// TwinCAT 3 PLC project PLC01
// ProgramVersion: 3.1.4024.0
// libraries:
//   Tc2_Standard, * (Beckhoff Automation GmbH)
//   Tc2_System, * (Beckhoff Automation GmbH)
//   Tc2_Utilities, * (Beckhoff Automation GmbH)
//   Tc3_Database, * (Beckhoff Automation GmbH)
//   Tc3_EventLogger, * (Beckhoff Automation GmbH)
//   Tc3_Module, * (Beckhoff Automation GmbH)
// project tree:
//   DUTs/Database/ ST_DatabasePower.TcDUT
//   DUTs/HMI/ ST_Valve.TcDUT
//   DUTs/PowerMeter/ ST_AuxConvertedMeasure.TcDUT, ST_AuxiliaryPowerValues.TcDUT, ST_Channel.TcDUT, ST_ConvertedPower.TcDUT, ST_PowerMeter.TcDUT
//   DUTs/ ST_Convert.TcDUT
//   FBs/Database/General/ FB_SQL_ExecuteComandWithoutReturn.TcPOU, FB_SQL_ReadWithData.TcPOU, FB_SQL_TO_CSV.TcPOU
//   FBs/Database/PowerMeter/ FB_SQL_ReadPower.TcPOU, FB_SQL_WritePower.TcPOU
//   FBs/PowerMeter/ FB_LastTimeSimple.TcPOU, FB_MeasureAuxPhasePower.TcPOU, FB_PowerMeter.TcPOU, FB_Simulate_EL3433.TcPOU
//   FBs/Process/ FB_Pump.TcPOU, FB_Valve.TcPOU
//   FCs/ FC_ConcatStr.TcPOU
//   GVLs/ GVL.TcGVL, GVL_HMI.TcGVL, GVL_IO.TcGVL
//   / PlcTask.TcTTO
//   POUs/Database/ PRG_Database.TcPOU
//   POUs/Eletric/ PRG_Eletric.TcPOU
//   POUs/ MAIN.TcPOU
//   POUs/PowerMeter/ PRG_PowerMeter.TcPOU
//   POUs/Process/ PRG_Process.TcPOU
// real-time tasks:
//   TASK PlcTask: cycle T#10ms, priority 20, ADS port 350
// motion (NC):
//   TASK NC-Task 1 SAF: cycle T#2ms, priority 4, ADS port 501
//   TASK NC-Task 1 SVB: cycle T#10ms, priority 8, ADS port 511
//   AXIS Eixo X (id 1)
//     OtherSettings: AllowMotionCmdToSlave=true
//     encoder EncType=1
//     drive DrvType=5
//       Analog: TorqueSetpointScale=10, ScaleFactorActTorque=0.1
//     controller CtrType=1
//       CtrPara: PriorControlFactor=1
//         Observer: BandWidth=20
// I/O:
//   DEVICE Device 3 (EtherCAT), AmsNetId 169.254.242.29.4.1
//     Term 1 (EK1100) [EK1100 EtherCAT Coupler (2A E-Bus)]
//       Term 2 (EL1008) [EL1008 8Ch. Dig. Input 24V, 3ms]
//       Term 3 (EL2008) [EL2008 8Ch. Dig. Output 24V, 0.5A]
//       Term 4 (EL3062) [EL3062 2Ch. Ana. Input 0-10V]
//       Term 5 (EL4002) [EL4002 2Ch. Ana. Output 0-10V, 12bit]
//       Term 6 (EL3433) [EL3433 3Ch. Power Measuring]
//       Term 7 (EL6900) [EL6900, TwinSAFE PLC]
//       Term 8 (EK1310) [EK1310 EtherCAT P extension with feed-in]
// variable links:
//   PLC01/PLC01 Instance <-> Device 3 (EtherCAT)/Term 1 (EK1100)/Term 6 (EL3433)
//     PlcTask Inputs/PRG_PowerMeter.EL3433_Ch1/ActivePower <-> PM Inputs Channel 1/Active power
//     PlcTask Inputs/PRG_PowerMeter.EL3433_Ch2/ActivePower <-> PM Inputs Channel 2/Active power
//     PlcTask Inputs/PRG_PowerMeter.EL3433_Ch3/ActivePower <-> PM Inputs Channel 3/Active power
//     PlcTask Inputs/PRG_PowerMeter.EL3433_Ch1/Current <-> PM Inputs Channel 1/Current
//     PlcTask Inputs/PRG_PowerMeter.EL3433_Ch2/Current <-> PM Inputs Channel 2/Current
//     PlcTask Inputs/PRG_PowerMeter.EL3433_Ch3/Current <-> PM Inputs Channel 3/Current
//     PlcTask Inputs/PRG_PowerMeter.EL3433_Ch1/Index <-> PM Inputs Channel 1/Index
//     PlcTask Inputs/PRG_PowerMeter.EL3433_Ch2/Index <-> PM Inputs Channel 2/Index
//     PlcTask Inputs/PRG_PowerMeter.EL3433_Ch3/Index <-> PM Inputs Channel 3/Index
//     PlcTask Inputs/PRG_PowerMeter.EL3433_Ch1/Status/MissingZeroCrossing <-> PM Inputs Channel 1/STATUS/Missing zero crossing
//     PlcTask Inputs/PRG_PowerMeter.EL3433_Ch2/Status/MissingZeroCrossing <-> PM Inputs Channel 2/STATUS/Missing zero crossing
//     PlcTask Inputs/PRG_PowerMeter.EL3433_Ch3/Status/MissingZeroCrossing <-> PM Inputs Channel 3/STATUS/Missing zero crossing
//     PlcTask Inputs/PRG_PowerMeter.EL3433_Ch1/Status/OverCurrent <-> PM Inputs Channel 1/STATUS/Overcurrent
//     PlcTask Inputs/PRG_PowerMeter.EL3433_Ch2/Status/OverCurrent <-> PM Inputs Channel 2/STATUS/Overcurrent
//     PlcTask Inputs/PRG_PowerMeter.EL3433_Ch3/Status/OverCurrent <-> PM Inputs Channel 3/STATUS/Overcurrent
//     PlcTask Inputs/PRG_PowerMeter.EL3433_Ch1/Status/OverVoltage <-> PM Inputs Channel 1/STATUS/Overvoltage
//     PlcTask Inputs/PRG_PowerMeter.EL3433_Ch2/Status/OverVoltage <-> PM Inputs Channel 2/STATUS/Overvoltage
//     PlcTask Inputs/PRG_PowerMeter.EL3433_Ch3/Status/OverVoltage <-> PM Inputs Channel 3/STATUS/Overvoltage
//     PlcTask Inputs/PRG_PowerMeter.EL3433_Ch1/Status/PhaseSeqCCW <-> PM Inputs Channel 1/STATUS/Phase sequence ccw
//     PlcTask Inputs/PRG_PowerMeter.EL3433_Ch2/Status/PhaseSeqCCW <-> PM Inputs Channel 2/STATUS/Phase sequence ccw
//     PlcTask Inputs/PRG_PowerMeter.EL3433_Ch3/Status/PhaseSeqCCW <-> PM Inputs Channel 3/STATUS/Phase sequence ccw
//     PlcTask Inputs/PRG_PowerMeter.EL3433_Ch1/Status/PhaseSeqCW <-> PM Inputs Channel 1/STATUS/Phase sequence cw
//     PlcTask Inputs/PRG_PowerMeter.EL3433_Ch2/Status/PhaseSeqCW <-> PM Inputs Channel 2/STATUS/Phase sequence cw
//     PlcTask Inputs/PRG_PowerMeter.EL3433_Ch3/Status/PhaseSeqCW <-> PM Inputs Channel 3/STATUS/Phase sequence cw
//     PlcTask Inputs/PRG_PowerMeter.EL3433_Ch1/Status/TxPdoState <-> PM Inputs Channel 1/STATUS/TxPDO State
//     PlcTask Inputs/PRG_PowerMeter.EL3433_Ch2/Status/TxPdoState <-> PM Inputs Channel 2/STATUS/TxPDO State
//     PlcTask Inputs/PRG_PowerMeter.EL3433_Ch3/Status/TxPdoState <-> PM Inputs Channel 3/STATUS/TxPDO State
//     PlcTask Inputs/PRG_PowerMeter.EL3433_Ch1/Status/TxPdoToggle <-> PM Inputs Channel 1/STATUS/TxPDO Toggle
//     PlcTask Inputs/PRG_PowerMeter.EL3433_Ch2/Status/TxPdoToggle <-> PM Inputs Channel 2/STATUS/TxPDO Toggle
//     PlcTask Inputs/PRG_PowerMeter.EL3433_Ch3/Status/TxPdoToggle <-> PM Inputs Channel 3/STATUS/TxPDO Toggle
//     PlcTask Inputs/PRG_PowerMeter.EL3433_Ch1/Status/UnderVoltage <-> PM Inputs Channel 1/STATUS/Undervoltage
//     PlcTask Inputs/PRG_PowerMeter.EL3433_Ch2/Status/UnderVoltage <-> PM Inputs Channel 2/STATUS/Undervoltage
//     PlcTask Inputs/PRG_PowerMeter.EL3433_Ch3/Status/UnderVoltage <-> PM Inputs Channel 3/STATUS/Undervoltage
//     PlcTask Inputs/PRG_PowerMeter.EL3433_Ch1/VariantValue <-> PM Inputs Channel 1/Variant value
//     PlcTask Inputs/PRG_PowerMeter.EL3433_Ch2/VariantValue <-> PM Inputs Channel 2/Variant value
//     PlcTask Inputs/PRG_PowerMeter.EL3433_Ch3/VariantValue <-> PM Inputs Channel 3/Variant value
//     PlcTask Inputs/PRG_PowerMeter.EL3433_Ch1/Voltage <-> PM Inputs Channel 1/Voltage
//     PlcTask Inputs/PRG_PowerMeter.EL3433_Ch2/Voltage <-> PM Inputs Channel 2/Voltage
//     PlcTask Inputs/PRG_PowerMeter.EL3433_Ch3/Voltage <-> PM Inputs Channel 3/Voltage
//     PlcTask Outputs/PRG_PowerMeter.Ch1_OutIndex <-> PM Outputs Channel 1/Index
//     PlcTask Outputs/PRG_PowerMeter.Ch2_OutIndex <-> PM Outputs Channel 2/Index
//     PlcTask Outputs/PRG_PowerMeter.Ch3_OutIndex <-> PM Outputs Channel 3/Index
//     PlcTask Outputs/PRG_PowerMeter.ChAux_OutIndex <-> PM Outputs Auxiliary/Index

CONFIGURATION PLC01
    RESOURCE PLC ON TwinCAT3
        TASK PlcTask(INTERVAL := T#10ms, PRIORITY := 20);
        PROGRAM MAIN WITH PlcTask : MAIN;
    END_RESOURCE
END_CONFIGURATION

// ---- DUTs/Database/ST_DatabasePower.TcDUT
TYPE ST_DatabasePower :
STRUCT
	ID 					: T_ULARGE_INTEGER  ;	//IDENTITY
	Timestamp 			: DATE_AND_TIME ;		//TIMESTAMP
	Name 				: STRING(50) ;			//NAME OF LOAD
	ActivePower 		: LREAL ;				//ACTIVE POWER
	ApparentPower 		: LREAL ;				//APARENT POWER
	ReactivePower 		: LREAL ;				//REACTIVE POWER
	Voltage 			: LREAL ;				//VOLTAGE
	Current 			: LREAL ;				//CURRENT
	Cosphi				: LREAL	;				//COSENO PHI
	Frequency			: LREAL	;				//FREQUENCY
	AngleBetweenPhase1	: LREAL	;				//ANGLE BETWEEN FASE 1	
	Energy 				: LREAL ;				//POSITIVE ENERGY
	EnergyNegative		: LREAL	;				//NEGATIVE ENERGY
END_STRUCT
END_TYPE

// ---- DUTs/HMI/ST_Valve.TcDUT
TYPE ST_Valve :
STRUCT
	status : BOOL ;
	comando : BOOL ;
	auto_manual : BOOL ;
	time_feedback : INT ;
END_STRUCT
END_TYPE

// ---- DUTs/PowerMeter/ST_AuxConvertedMeasure.TcDUT
TYPE ST_AuxConvertedMeasure :
	STRUCT
		sumOfEnergy : LREAL;									//index 2. 
		frequency : LREAL;										//4
		sumOfEnergyNeg : LREAL;									//5
		sumOfActivePower : LREAL;								//10
		sumOfApparentPower : LREAL;								//11
		sumOfReactivePower : LREAL;								//12
		adcTemp : LREAL ;										//100
		aHarmonicCurrentValue : ARRAY[1..3,1..21] OF LREAL;		//
		aHarmonicCurrentRatio : ARRAY[1..3,1..21] OF LREAL;		//
		aHarmonicVoltageValue : ARRAY[1..3,1..21] OF LREAL;		//
		aHarmonicVoltageRatio : ARRAY[1..3,1..21] OF LREAL;		//
		aAuxPowerValues : ARRAY[1..3] OF ST_ConvertedPower;		//
	END_STRUCT
END_TYPE

// ---- DUTs/PowerMeter/ST_AuxiliaryPowerValues.TcDUT
TYPE ST_AuxiliaryPowerValues :
	STRUCT
		index:USINT;		//Indice
		channel:USINT;		//Canal
		value:DINT;			//Valor
	END_STRUCT
END_TYPE

// ---- DUTs/PowerMeter/ST_Channel.TcDUT
TYPE ST_Channel :
	STRUCT
		OverVoltage : BIT ; //
		UnderVoltage : BIT ; //
		OverCurrent : BIT ; //
		PhaseSeqCW : BIT ; //
		PhaseSeqCCW : BIT ; //
		MissingZeroCrossing : BIT ; //
		TxPdoState : BIT ; //
		TxPdoToggle : BIT ; //
	END_STRUCT
END_TYPE

// ---- DUTs/PowerMeter/ST_ConvertedPower.TcDUT
TYPE ST_ConvertedPower :
	STRUCT
		Current			:LREAL	;	//Display the channel's current 
		Voltage			:LREAL	;	//Display the channel's voltage
		ActivePower		:LREAL	;	//Display the channel's active power
		ApparentPower	:LREAL	;	//Potência aparente
		ReactivePower	:LREAL	;	//potencia reativa
		Energy			:LREAL	;	//Energia
		Cosphi			:LREAL	;	//cosseno PHI
		Frequency		:LREAL	;	//Display the channel's Frequency
		EnergyNegative	:LREAL	;	//Energia (Negativa)
		AngleBetweenPhase1	:LREAL	;	//Angulo entre essa fase e a fase 1
	END_STRUCT
END_TYPE

// ---- DUTs/PowerMeter/ST_PowerMeter.TcDUT
TYPE ST_PowerMeter :
	STRUCT
		Status 			: ST_Channel ; 	//Todos os status de cada canal (Overvoltage, UnderVoltage, Overcurrent, PhaseSequenceZero Crossing...)
		Current 		: DINT ; 		//
		Voltage 		: DINT ; 		//
		ActivePower 	: DINT ; 		//
		Index 			: USINT ; 		//
		VariantValue	: DINT ; 		//
	END_STRUCT
END_TYPE

// ---- DUTs/ST_Convert.TcDUT
TYPE ST_Convert :
UNION
	aWORD : ARRAY[0..10] OF INT ;
	aREAL : ARRAY[0..5] OF REAL ;
END_UNION
END_TYPE

// ---- GVLs/GVL.TcGVL
{attribute 'qualified_only'}
VAR_GLOBAL
	(* Estruturas com os valores convertidos *)	
	EL3433_Ch1_PowerConverted : ST_ConvertedPower; //Estrutura que retorna os valores da Fase 1 (Tensao, Corrente...)
	EL3433_Ch2_PowerConverted : ST_ConvertedPower; //Estrutura que retorna os valores da Fase 1 (Tensao, Corrente...)
	EL3433_Ch3_PowerConverted : ST_ConvertedPower; //Estrutura que retorna os valores da Fase 1 (Tensao, Corrente...)
END_VAR

// ---- GVLs/GVL_HMI.TcGVL
{attribute 'qualified_only'}
VAR_GLOBAL
	DateStart : STRING ;
	DateEnd : STRING ;
END_VAR

// ---- GVLs/GVL_IO.TcGVL
{attribute 'qualified_only'}
VAR_GLOBAL


END_VAR

// ---- POUs/MAIN.TcPOU
PROGRAM MAIN
VAR
	stMyTest : ST_Convert ;

END_VAR



PRG_PowerMeter() ;

PRG_Database();

END_PROGRAM

// ---- POUs/PowerMeter/PRG_PowerMeter.TcPOU
PROGRAM PRG_PowerMeter
VAR	

(* Seleciona vaores REAIS do EL3433 ou Simulados *)
	bSelectValues : BOOL ;

(* Bloco para simulacao de valores do EL3433 *)
	fbPowerL1Simulate : FB_Simulate_EL3433 ;
	fbPowerL2Simulate : FB_Simulate_EL3433 ;
	fbPowerL3Simulate : FB_Simulate_EL3433 ;

(* Blocos de funcao para cada canal do terminal EL3433 REAL *)	
	fbPowerL1 : FB_PowerMeter ; //Bloco para extratir os dados do cartão
	fbPowerL2 : FB_PowerMeter ; //Bloco para extratir os dados do cartão
	fbPowerL3 : FB_PowerMeter ; //Bloco para extratir os dados do cartão
	fbAuxPower : FB_MeasureAuxPhasePower ; //	
	
(* Estruturas com link com o IO EL3433*)
	EL3433_Ch1 AT %I* : ST_PowerMeter ;
	EL3433_Ch2 AT %I* : ST_PowerMeter ;
	EL3433_Ch3 AT %I* : ST_PowerMeter ;	

(* Variavel Index do terminal EL3433 *)
	Ch1_OutIndex AT %Q*: USINT := 0 ;
	Ch2_OutIndex AT %Q*: USINT := 0 ;
	Ch3_OutIndex AT %Q*: USINT := 0 ;
	ChAux_OutIndex AT %Q*: USINT := 0 ;	
	

	stConvertedAuxChn : ST_AuxConvertedMeasure; //	
	
END_VAR


IF bSelectValues = FALSE THEN
	
	fbPowerL1Simulate(
		bExecute:= TRUE, 
		Current=> GVL.EL3433_Ch1_PowerConverted.Current, 
		Voltage=> GVL.EL3433_Ch1_PowerConverted.Voltage, 
		ActivePower=> GVL.EL3433_Ch1_PowerConverted.ActivePower, 
		ApparentPower=> GVL.EL3433_Ch1_PowerConverted.ApparentPower, 
		ReactivePower=> GVL.EL3433_Ch1_PowerConverted.ReactivePower, 
		Energy=> GVL.EL3433_Ch1_PowerConverted.Energy, 
		Cosphi=> GVL.EL3433_Ch1_PowerConverted.Cosphi, 
		Frequency=> GVL.EL3433_Ch1_PowerConverted.Frequency, 
		EnergyNegative=> GVL.EL3433_Ch1_PowerConverted.EnergyNegative, 
		AngleBetweenPhase1=> GVL.EL3433_Ch1_PowerConverted.AngleBetweenPhase1);
		
		
		GVL.EL3433_Ch2_PowerConverted := GVL.EL3433_Ch1_PowerConverted;
		GVL.EL3433_Ch3_PowerConverted := GVL.EL3433_Ch1_PowerConverted;
ELSE

	fbPowerL1(PowerInput:= EL3433_Ch1, PowerConverted=> GVL.EL3433_Ch1_PowerConverted, OutIndex=> Ch1_OutIndex);
	fbPowerL2(PowerInput:= EL3433_Ch2, PowerConverted=> GVL.EL3433_Ch2_PowerConverted, OutIndex=> Ch2_OutIndex);
	fbPowerL3(PowerInput:= EL3433_Ch3, PowerConverted=> GVL.EL3433_Ch3_PowerConverted, OutIndex=> Ch3_OutIndex);
	fbAuxPower(convertedMeasure=> stConvertedAuxChn);


END_IF

END_PROGRAM

// ---- FBs/PowerMeter/FB_Simulate_EL3433.TcPOU
FUNCTION_BLOCK FB_Simulate_EL3433
VAR_INPUT
	bExecute : BOOL ;
END_VAR
VAR_OUTPUT
	Current			:LREAL	;	//Display the channel's current 
	Voltage			:LREAL	;	//Display the channel's voltage
	ActivePower		:LREAL	;	//Display the channel's active power
	ApparentPower	:LREAL	;	//Potência aparente
	ReactivePower	:LREAL	;	//potencia reativa
	Energy			:LREAL	;	//Energia
	Cosphi			:LREAL	;	//cosseno PHI
	Frequency		:LREAL	;	//Display the channel's Frequency
	EnergyNegative	:LREAL	;	//Energia (Negativa)
	AngleBetweenPhase1	:LREAL	;	//Angulo entre essa fase e a fase 1
END_VAR
VAR
    tCurrentTime: TIME;
    rRandomValue: REAL;
	fRandom : DRAND ;
END_VAR


   fRandom(Seed:= 1 , Num=> rRandomValue);  // Converte o tempo atual para milissegundos

IF bExecute = TRUE THEN 

	Current			:=	rRandomValue + 2;	//Display the channel's current 
	Voltage			:=	rRandomValue + 379;	//Display the channel's voltage
	Cosphi			:=	(rRandomValue + 81) * 0.01;		
	ActivePower		:=	Voltage * Current * Cosphi;	//Display the channel's active power
	ApparentPower	:=	Voltage * Current;	//Potência aparente
	ReactivePower	:=	Voltage * Current * SQRT( 1 - Cosphi * Cosphi) ;	//potencia reativa
	Energy			:=	rRandomValue * 10;	
	Frequency		:=	rRandomValue + 59;	
	EnergyNegative	:=	rRandomValue * 10;	
	AngleBetweenPhase1	:=	rRandomValue + 60;	
END_IF

END_FUNCTION_BLOCK

// ---- FBs/PowerMeter/FB_PowerMeter.TcPOU
FUNCTION_BLOCK FB_PowerMeter
VAR_INPUT
	PowerInput : ST_PowerMeter;	
END_VAR
VAR_OUTPUT
	PowerConverted : ST_ConvertedPower;	//Valores convertidos
	OutIndex : USINT :=0;	
END_VAR
VAR
	iAux:UINT:=0;
END_VAR

(* Conversao da corrente *)
powerConverted.current:=DINT_TO_LREAL(PowerInput.current)*0.000001;

(* Conversao da Tensao *)
powerConverted.voltage:=DINT_TO_LREAL(PowerInput.voltage)*0.0001;

(* Conversao da potencia ativa *)
powerConverted.activePower:=DINT_TO_LREAL(PowerInput.activePower)*0.01;

(* Conversoes diversas *)

CASE PowerInput.index OF
	0:
		powerConverted.apparentPower := DINT_TO_LREAL(PowerInput.variantValue) * 0.01 ;
	1:
		powerConverted.reactivePower := DINT_TO_LREAL(PowerInput.variantValue) * 0.01 ;
	2:
		powerConverted.energy := DINT_TO_LREAL(PowerInput.variantValue) * 0.001;
	3:
		powerConverted.cosphi := DINT_TO_LREAL(PowerInput.variantValue) * 0.001;
	4:
		powerConverted.frequency := DINT_TO_LREAL(PowerInput.variantValue) * 0.1;
	5:
		powerConverted.energy := DINT_TO_LREAL(PowerInput.variantValue) * 0.001 ;
	6:
		powerConverted.AngleBetweenPhase1 := DINT_TO_LREAL(PowerInput.variantValue) * 0.01;
END_CASE

IF (PowerInput.index = OutIndex)THEN
	iAux := iAux + 1 ;
	IF iAux > 4 THEN
		iAux := 0 ;
		IF outIndex <= 6 THEN
			outIndex := outIndex + 1 ;
		ELSE
			outIndex := 0 ;	
		END_IF
	END_IF	
END_IF

END_FUNCTION_BLOCK

// ---- FBs/PowerMeter/FB_MeasureAuxPhasePower.TcPOU
FUNCTION_BLOCK FB_MeasureAuxPhasePower
VAR_INPUT
END_VAR
VAR_OUTPUT
	convertedMeasure:ST_AuxConvertedMeasure;
	tLastHarmonicMeasureTime:TIME;
	lastiTime:FB_LastTimeSimple;
END_VAR
VAR
	power AT %I*:ST_AuxiliaryPowerValues;
	iChannel AT %Q*:USINT;
	iIndex AT %Q*:USINT;
	bMeasureTime:BOOL;
END_VAR

CASE power.channel OF
	0:
		CASE power.index OF
			0:
				iIndex := 2 ;
			2:
				convertedMeasure.sumOfEnergy := DINT_TO_LREAL(power.value) * 0.001;
				iIndex:=4;
				//F_DebugCount(1);
			4:
				convertedMeasure.frequency := DINT_TO_LREAL(power.value) * 0.1;
				iIndex:=5;
				//F_DebugCount(2);
			5:
				convertedMeasure.sumOfEnergyNeg := DINT_TO_LREAL(power.value) * 0.001;
				iIndex:=10;
				//F_DebugCount(3);				
			10:
				convertedMeasure.sumOfActivePower := DINT_TO_LREAL(power.value) * 0.01;
				iIndex:=11;
				//F_DebugCount(4);
			11:
				convertedMeasure.sumOfApparentPower := DINT_TO_LREAL(power.value)*0.01;
				iIndex:=12;
				//F_DebugCount(5);				
			12:
				convertedMeasure.sumOfReactivePower := DINT_TO_LREAL(power.value)*0.01;
				iIndex:=100;
				//F_DebugCount(6);				
			100:
				convertedMeasure.adcTemp := DINT_TO_LREAL(power.value);
				iIndex:=1;
				iChannel:=1;
				bMeasureTime:=TRUE;	//Inicia o tempo de leitura das harmonicas
				//F_DebugCount(7);
		END_CASE
	1..3:
		CASE power.index OF
			0:
				;
			100:
				;
			1..21:
				convertedMeasure.aHarmonicCurrentValue[power.channel,power.index]:=DINT_TO_LREAL(power.value)*0.000001;
				IF (power.index <21) AND (iIndex < 21) THEN
					iIndex:=iIndex+1;
				ELSIF (power.index = 21 ) AND (power.channel < 3) THEN
					iIndex:=1;
					IF power.channel = iChannel THEN
						iChannel:=iChannel+1;
					END_IF
				ELSIF (power.index = 21) AND (power.channel >=3) THEN
					iChannel:=1;		//Modificar
					iIndex:=51;
				END_IF
			51..71:
				convertedMeasure.aHarmonicCurrentRatio[power.channel,power.index-50]:=DINT_TO_LREAL(power.value)*0.01;
				IF (power.index <71) AND (iIndex < 71) THEN
					iIndex:=iIndex+1;
				ELSIF (power.index = 71 ) AND (power.channel < 3) THEN
					iIndex:=51;
					IF power.channel = iChannel THEN
						iChannel:=iChannel+1;
					END_IF
				ELSIF (power.index = 71) AND (power.channel >=3) THEN
					iChannel:=1;		//Modificar
					iIndex:=101;
				END_IF
			101..121:
				convertedMeasure.aHarmonicVoltageValue[power.channel,power.index-100]:=DINT_TO_LREAL(power.value)*0.0001;
				IF (power.index <121) AND (iIndex < 121) THEN
					iIndex:=iIndex+1;
				ELSIF (power.index = 121 ) AND (power.channel < 3) THEN
					iIndex:=101;
					IF power.channel = iChannel THEN
						iChannel:=iChannel+1;
					END_IF
				ELSIF (power.index = 121) AND (power.channel >=3) THEN
					iChannel:=1;		//Modificar
					iIndex:=151;
				END_IF

			151..171:
				convertedMeasure.aHarmonicVoltageRatio[power.channel,power.index-150]:=DINT_TO_LREAL(power.value)*0.01;
				IF (power.index <171) AND (iIndex < 171) THEN
					iIndex:=iIndex+1;
				ELSIF (power.index = 171 ) AND (power.channel < 3) THEN
					iIndex:=151;
					IF power.channel = iChannel THEN
						iChannel:=iChannel+1;
					END_IF
				ELSIF (power.index = 171) AND (power.channel >=3) THEN
					iChannel:=11;		
					iIndex:=0;
					bMeasureTime:=FALSE;					
				END_IF
			ELSE
				iChannel:=0;
				iIndex:=0;
				bMeasureTime:=FALSE;
		END_CASE
	11..13:
		CASE power.index OF
			0:
				IF iIndex = power.index THEN
					iIndex := iIndex+1;
				END_IF
				convertedMeasure.aAuxPowerValues[power.channel-10].apparentPower := DINT_TO_LREAL(power.value)*0.01;
			1:
				IF iIndex = power.index THEN
					iIndex:=iIndex+1;
				END_IF	
				convertedMeasure.aAuxPowerValues[power.channel-10].reactivePower := DINT_TO_LREAL(power.value)*0.01;
			2:
				IF iIndex = power.index THEN
					iIndex:=iIndex+1;
				END_IF
				convertedMeasure.aAuxPowerValues[power.channel-10].energy := DINT_TO_LREAL(power.value)*0.001;
			3:
				IF iIndex = power.index THEN
					iIndex:=iIndex+1;
				END_IF
				convertedMeasure.aAuxPowerValues[power.channel-10].cosPhi := DINT_TO_LREAL(power.value)*0.001;
			4:
				IF iIndex = power.index THEN
					iIndex:=iIndex+1;
				END_IF
				convertedMeasure.aAuxPowerValues[power.channel-10].frequency := DINT_TO_LREAL(power.value)*0.1;
			5:
				IF iIndex = power.index THEN
					iIndex:=iIndex+1;
				END_IF
				convertedMeasure.aAuxPowerValues[power.channel-10].EnergyNegative := DINT_TO_LREAL(power.value)*0.001;
			6:
				IF iIndex = power.index THEN
					iIndex:=10;
				END_IF
				convertedMeasure.aAuxPowerValues[power.channel-10].AngleBetweenPhase1 := DINT_TO_LREAL(power.value)*0.01;
			10:
				IF iIndex = power.index THEN
					iIndex:=11;
				END_IF
				convertedMeasure.aAuxPowerValues[power.channel-10].current := DINT_TO_LREAL(power.value)*0.000001;
			11:
				IF iIndex = power.index THEN
					iIndex:=12;
				END_IF
				convertedMeasure.aAuxPowerValues[power.channel-10].voltage := DINT_TO_LREAL(power.value)*0.0001;
			12:
				convertedMeasure.aAuxPowerValues[power.channel-10].activePower := DINT_TO_LREAL(power.value)*0.01;
				IF power.channel = 13 THEN
					iIndex:=0;
					iChannel:=0;
				ELSE
					IF iChannel = power.channel AND power.channel < 13 THEN
						iChannel:=iChannel+1;
					END_IF
					iIndex:=0;
				END_IF
		END_CASE
END_CASE
lastiTime(bCountTime:= bMeasureTime, tLastTime=> tLastHarmonicMeasureTime);

END_FUNCTION_BLOCK

// ---- FBs/PowerMeter/FB_LastTimeSimple.TcPOU
FUNCTION_BLOCK FB_LastTimeSimple
VAR_INPUT
	bCountTime:BOOL;
END_VAR
VAR_OUTPUT
	tLastTime:TIME;
END_VAR
VAR
	t1:TON;
	timeCountedF_TRIG:F_TRIG;
	tActualtime:TIME;
END_VAR

IF timeCountedF_TRIG.Q THEN
	tLastTime:=tActualtime;
	tActualtime:=T#0S;
END_IF
timeCountedF_TRIG(CLK:=bCountTime);
t1(IN:= bCountTime, PT:=T#1D);
tActualtime:= MAX(tActualtime,t1.ET);

END_FUNCTION_BLOCK

// ---- POUs/Database/PRG_Database.TcPOU
PROGRAM PRG_Database
VAR
(* CREATE TABLE *)	
	fbCreateTable : FB_SQL_ExecuteComandWithoutReturn ;
	bCreateDatabase : BOOL ;
	bDatabaseCreated : BOOL ;
	sSqlCmdCreateTable : STRING(512) ;
	sError : STRING ;
	
(* CREATE CSV *)	
	fbSqlToCsv : FB_SQL_ExecuteComandWithoutReturn ;	
	sSqlCmdSqlToCsv : STRING(512) ;
	
(* WRITE TO DATABASE *)	
	fbSQLWrite_01 : FB_SQL_WritePower ;
	fbSQLWrite_02 : FB_SQL_WritePower ;
	fbSQLWrite_03 : FB_SQL_WritePower ;	
	bEnableWrite: BOOL := TRUE ;
	
(* READ FROM DATABASE *)	
	fbSQLRead_01 : FB_SQL_ReadPower ;
	

	bExecuteRead: BOOL;


END_VAR

(**********************************************************************************)	
(***************** CRIAR TABELA / CREATE TABLE / CREAR TABLA **********************)

sSqlCmdCreateTable := 'CREATE TABLE [TB_PowerMeter22] ([ID] bigint IDENTITY(1,1), [Timestamp] datetime, [Name] varchar(50), [ActivePower] float, [ApparentPower] float, [ReactivePower] float, [Voltage] float, [Current] float, [Cosphi] float, [Frequency] float, [AngleBetweenPhase1] float, [Energy] float, [EnergyNegative] float)';


IF 	M_CreateDatabase(bExecute:= bCreateDatabase, hDBID:= 1, sCommandSql:= sSqlCmdCreateTable ) THEN
;	
END_IF


(*
fbCreateTable(bExecute:= bCreateDatabase, 
			  hDBID:= 1, 
			  sCommandSql:= sSqlCmdCreateTable, 
			  bCommandOk=> bDatabaseCreated,
			  sError => sError);
*)
			  
(**********************************************************************************)			  
(*  ESCREVER NO BANCO DE DADOS A CADA 10S / WRITE TO DATABASE EVERY 10S/ ESCRIBIR EN LA BASE DE DATOS A CADA 10S *)

fbSQLWrite_01(
	sTableName:= 'TB_PowerMeter', 
	sNameLoad:= 'EL3433 CH1', 
	stEnergy:= GVL.EL3433_Ch1_PowerConverted, 
	bEnableWriteDatabase:= bEnableWrite, 
	iTimeWriteDatabase:= 10);
	
fbSQLWrite_02(
	sTableName:= 'TB_PowerMeter', 
	sNameLoad:= 'EL3433 CH2', 
	stEnergy:= GVL.EL3433_Ch2_PowerConverted, 
	bEnableWriteDatabase:= bEnableWrite, 
	iTimeWriteDatabase:= 10);

fbSQLWrite_03(
	sTableName:= 'TB_PowerMeter', 
	sNameLoad:= 'EL3433 CH3', 
	stEnergy:= GVL.EL3433_Ch3_PowerConverted, 
	bEnableWriteDatabase:= bEnableWrite, 
	iTimeWriteDatabase:= 10);	

	
	
(**********************************************************************************)			
(****** LER DO BANCO DE DADOS / READ FROM DATABASE / LEER DE LA BASE DE DATOS *****)	
	

GVL_HMI.DateStart:= '2023-07-25T16:08:14.020Z';
GVL_HMI.DateEnd := '2023-07-25T16:12:14.020Z';

fbSQLRead_01(
	bExecute:= bExecuteRead, 
	sTableName:= 'TB_PowerMeter', 
	sDateStart:= GVL_HMI.DateStart, 
	sDateEnd:= GVL_HMI.DateEnd, 
	bDone=> , 
	bBusy=> , 
	bError=> , 
	nRecords=> , 
	DataRead=> );	
	
	
	
(**********************************************************************************)		
(* GERAR CSV *)

sSqlCmdSQLToCSV := 'DECLARE @SQLQuery AS NVARCHAR(200) 
				DECLARE @FilePath AS NVARCHAR(200)  
				SET @SQLQuery = $'SELECT * FROM [DB_PowerMeasure].[dbo].[TB_PowerMeter]$'
				SET @FilePath = $'C:\temp\arquivo.csv$' 
				SET @SQLQuery = $'bcp "$' + @SQLQuery + $'" queryout "$' + @FilePath + $'" -c -t, -T -S DOUGLASC-NB01\SQLEXPRESS$'  
				EXEC xp_cmdshell @SQLQuery  ';

METHOD PUBLIC M_CreateDatabase : BOOL
VAR_INPUT
	bExecute : BOOL ;
	hDBID : INT ;
	sCommandSql : STRING(512) ;
END_VAR

VAR
	fbPulse: R_TRIG;
	fbSqlDatabase : FB_SQLDatabaseEvt(sNetID := '', tTimeout := T#10S);
	fbSqlCommand : FB_SQLCommandEvt(sNetID := '', tTimeout := T#180S) ;
    tcMessage    : I_TcMessage;	
	nState: INT;
END_VAR
fbPulse(CLK:= bExecute, Q=> );

IF fbPulse.Q THEN
	nState := 1 ;
END_IF

CASE nState OF
		
	0: (* Iddle *)
	;
	
	1:
	
	sError := '';
	nState := 10; 
	
	10: (* Connect to Database *)
	
	IF fbSqlDatabase.Connect(hDBID) THEN
		IF fbSqlDatabase.bError THEN
			nState := 250; 
        	tcMessage := fbSqlDatabase.ipTcResult;			
		ELSE
			nState := 20; 
		END_IF
	END_IF
	
	20:	(* Create Command *)
	
	IF fbSqlDatabase.CreateCmd(ADR(fbSqlCommand)) THEN
		IF fbSqlDatabase.bError THEN
			nState := 251; 
		ELSE
			nState := 30; 
		END_IF
	END_IF	
	
	30:  (* Execute Command *)
	
	IF fbSqlCommand.Execute(pSQLCmd:= ADR(sCommandSql), cbSQLCmd:= SIZEOF(sCommandSql)) THEN
		IF fbSQLCommand.bError THEN
			nState := 252; 
        	tcMessage := fbSQLCommand.ipTcResult;			
			M_CreateDatabase := FALSE ;			
		ELSE
			nState := 40; 
			M_CreateDatabase := TRUE ;
		END_IF
	END_IF	
	

	40:  (* Desconectar *)
	
	IF fbSqlDatabase.Disconnect() THEN
		IF fbSqlDatabase.bError THEN
			nState := 253;
		ELSE
			nState := 0;
   		END_IF
	END_IF

250: //Error step 10;
	sError := 'Erro no bloco Connect';
	nState := 40 ;

251: //Error step 20 ;
	sError := 'Erro no bloco Create Command';
	nState := 40 ;
252: //Error step 30 ;
	sError := 'Erro no bloco Execute Command';
	nState := 40 ;
253: //Error step 40 ;
	sError := 'Erro no bloco Disconect';
	nState := 40 ;
	
END_CASE
END_METHOD

END_PROGRAM

// ---- FBs/Database/General/FB_SQL_ExecuteComandWithoutReturn.TcPOU
FUNCTION_BLOCK FB_SQL_ExecuteComandWithoutReturn
VAR_INPUT
	bExecute : BOOL ;
	hDBID : UINT ;
	sCommandSql : STRING(512) ;
END_VAR
VAR_OUTPUT
	bCommandOk : BOOL ;
	sError : STRING ;
END_VAR
VAR
	fbSqlDatabase : FB_SQLDatabaseEvt(sNetID := '', tTimeout := T#10S);
	fbSqlCommand : FB_SQLCommandEvt(sNetID := '', tTimeout := T#180S) ;
    tcMessage    : I_TcMessage;	
	nState : INT ;
	fbPulse : R_TRIG ;
END_VAR

fbPulse(CLK:= bExecute, Q=> );

IF fbPulse.Q THEN
	nState := 1 ;
END_IF

CASE nState OF
		
	0: (* Iddle *)
	;
	
	1:
	
	sError := '';
	nState := 10; 
	
	10: (* Connect to Database *)
	
	IF fbSqlDatabase.Connect(hDBID) THEN
		IF fbSqlDatabase.bError THEN
			nState := 250; 
        	tcMessage := fbSqlDatabase.ipTcResult;			
		ELSE
			nState := 20; 
		END_IF
	END_IF
	
	20:	(* Create Command *)
	
	IF fbSqlDatabase.CreateCmd(ADR(fbSqlCommand)) THEN
		IF fbSqlDatabase.bError THEN
			nState := 251; 
		ELSE
			nState := 30; 
		END_IF
	END_IF	
	
	30:  (* Execute Command *)
	
	IF fbSqlCommand.Execute(pSQLCmd:= ADR(sCommandSql), cbSQLCmd:= SIZEOF(sCommandSql)) THEN
		IF fbSQLCommand.bError THEN
			nState := 252; 
        	tcMessage := fbSQLCommand.ipTcResult;			
			bCommandOk := FALSE ;			
		ELSE
			nState := 40; 
			bCommandOk := TRUE ;
		END_IF
	END_IF	
	

	40:  (* Desconectar *)
	
	IF fbSqlDatabase.Disconnect() THEN
		IF fbSqlDatabase.bError THEN
			nState := 253;
		ELSE
			nState := 0;
   		END_IF
	END_IF

250: //Error step 10;
	sError := 'Erro no bloco Connect';
	nState := 40 ;

251: //Error step 20 ;
	sError := 'Erro no bloco Create Command';
	nState := 40 ;
252: //Error step 30 ;
	sError := 'Erro no bloco Execute Command';
	nState := 40 ;
253: //Error step 40 ;
	sError := 'Erro no bloco Disconect';
	nState := 40 ;
	
END_CASE

END_FUNCTION_BLOCK

// ---- FBs/Database/PowerMeter/FB_SQL_WritePower.TcPOU
FUNCTION_BLOCK FB_SQL_WritePower
VAR_INPUT
	sTableName : T_MaxString;
	sNameLoad : STRING(50)	;
	dtTimestamp : DT;
	stEnergy : ST_ConvertedPower ;	
	bEnableWriteDatabase : BOOL;
	iTimeWriteDatabase : INT ;
END_VAR
VAR_OUTPUT
END_VAR
VAR
	ColumnInfo    	: ARRAY [0..12] OF ST_ColumnInfo;//Informações das colunas para criar tabela
	ColumnNames     :  ARRAY[0..12] OF STRING(50);//Nome das colunas para salvar dados
	DataToWrite 	: ST_DatabasePower ;
	Timer 	: TON;
    fbPLCDBWrite    :  FB_PLCDBWriteEvt(sNetID := '', tTimeout := T#5S); // Escrever dados
	tcMessageWrite       :  I_TcMessage;
	nRecords : UDINT ;
    systime         :	GETSYSTEMTIME;									 //Faz a leitura da data e hora do sistema
    currentTime     :	T_FILETIME;										 //
	
	
END_VAR

// Clock 10 segundos
Timer(IN:= NOT Timer.Q , PT:= TO_TIME(iTimeWriteDatabase*1000) , Q=> , ET=> );


//Date Time
systime(timeLoDw => currentTime.dwLowDateTime, timeHiDW => currentTime.dwHighDateTime );


//Dados.ID := 0;//Comentado pois assim o próprio SQL gera o ID único do dado;
DataToWrite.Timestamp := FILETIME_TO_DT(currentTime);
DataToWrite.Name := sNameLoad ;
DataToWrite.ActivePower := stEnergy.ActivePower;
DataToWrite.ApparentPower := stEnergy.ApparentPower;
DataToWrite.ReactivePower := stEnergy.ReactivePower;
DataToWrite.Voltage := stEnergy.Voltage;
DataToWrite.Current := stEnergy.Current;
DataToWrite.Cosphi := stEnergy.Cosphi;
DataToWrite.Frequency := stEnergy.Frequency;
DataToWrite.AngleBetweenPhase1 := stEnergy.AngleBetweenPhase1;
DataToWrite.Energy := stEnergy.Energy;
DataToWrite.EnergyNegative := stEnergy.EnergyNegative;



// Definição do nome das colunas
ColumnNames[0] := 'ID';
ColumnNames[1] := 'Timestamp';
ColumnNames[2] := 'Name';
ColumnNames[3] := 'ActivePower';
ColumnNames[4] := 'ApparentPower';
ColumnNames[5] := 'ReactivePower';
ColumnNames[6] := 'Voltage';
ColumnNames[7] := 'Current';
ColumnNames[8] := 'Cosphi';
ColumnNames[9] := 'Frequency';
ColumnNames[10] := 'AngleBetweenPhase1';
ColumnNames[11] := 'Energy';
ColumnNames[12] := 'EnergyNegative';


// Chamada da função de escrita
IF Timer.Q  THEN
	IF fbPLCDBWrite.WriteStruct(
		hDBID:= 1, 
		sTableName:= sTableName, 
		pRecord:= ADR(DataToWrite), 
		cbRecord:= SIZEOF(DataToWrite), 
		pColumnNames:= ADR(ColumnNames), 
		cbColumnNames:= SIZEOF(ColumnNames))
	THEN
		IF fbPLCDBWrite.bError THEN
			tcMessageWrite := fbPLCDBWrite.ipTcResult;
		END_IF
	END_IF 
END_IF

END_FUNCTION_BLOCK

// ---- FBs/Database/PowerMeter/FB_SQL_ReadPower.TcPOU
FUNCTION_BLOCK FB_SQL_ReadPower
VAR_INPUT
	bExecute : BOOL;
	sTableName : STRING;
	sDateStart : STRING;
	sDateEnd : STRING ;
END_VAR
VAR_OUTPUT
	bDone : BOOL;
	bBusy : BOOL;
	bError : BOOL;
	nRecords : UDINT;
	DataRead : ARRAY[0..10000] OF ST_DatabasePower;
END_VAR
VAR
	hDBID : UDINT 	:= 1;
	fbSqlDatabase : FB_SQLDatabaseEvt(sNetID := '', tTimeout := T#180S);
	fbSqlCommand : FB_SQLCommandEvt(sNetID := '', tTimeout := T#180S) ;
    fbSqlResult : FB_SQLResultEvt(sNetID:='', tTimeout    := T#180S); 
	sCommandSql  	: STRING (1500); //Comando SQL
	bRead 			: BOOL;	
	fbPulse : R_TRIG ;	
	sDateStartAux : STRING ;	
	sDateEndtAux : STRING ;	
	nState: INT;
	counter: INT;
END_VAR

// Tratamento da data e hora da STRING recebida da IHM
//sDateStartAux := REPLACE(STR1:= sDateStart, STR2:= ' ', L:= 1, P:= 11);
sDateStartAux := LEFT(sDateStart, 19);

//sDateEndtAux := REPLACE(STR1:= sDateEnd, STR2:= ' ', L:= 1, P:= 11);
sDateEndtAux := LEFT(sDateEnd, 19);
		

//Ejemplo comando SQL
//'SELECT * FROM TB_PowerMeasure WHERE Timestamp BETWEEN $'2023-06-27 00:00:00$' AND $'2023-06-27 17:00:00$' '


// Montagem do comando SQL		

sCommandSql := 'SELECT * FROM TB_PowerMeasure WHERE Timestamp BETWEEN $'';
sCommandSql := FC_ConcatStr(sCommandSql, sDateStartAux) ;
sCommandSql := FC_ConcatStr(sCommandSql, '$' AND $'') ;	
sCommandSql := FC_ConcatStr(sCommandSql, sDateEndtAux) ;	
sCommandSql := FC_ConcatStr(sCommandSql, '$'') ;	


//sCommandSql := 'SELECT TOP (1) *  FROM [DB_PowerMeasure].[dbo].[TB_PowerMeasure]';


// Pulso para comando SQL
fbPulse(CLK:= bExecute, Q=> );
IF fbPulse.Q = TRUE THEN
	nState := 1 ;
END_IF

counter := counter + 1 ;

CASE nState OF

	0:
	
		;
	
	
	1: 
	
	IF fbSqlDatabase.Disconnect() THEN
		IF fbSqlDatabase.bError THEN
			nState := 255;
		ELSE
			nState := 10;
   		END_IF
	END_IF
	
	nState := 1 ;
	
(* CONECTAR AO BANCO / CONNECT TO DATABASE / *)
	10:
	
	IF fbSqlDatabase.Connect(hDBID) THEN
		IF fbSqlDatabase.bError THEN
			nState := 250; 
		ELSE
			nState := 20; 
		END_IF
	END_IF
	
	20:	
	IF fbSqlDatabase.CreateCmd(ADR(fbSqlCommand)) THEN
		IF fbSqlDatabase.bError THEN
			nState := 251; 
		ELSE
			nState := 30; 
		END_IF
	END_IF	

	
	30:
	IF fbSqlCommand.ExecuteDataReturn(ADR(sCommandSql), SIZEOF(sCommandSql), ADR(fbSqlResult)) THEN
		IF fbSQLCommand.bError THEN
			nState := 252; 
		ELSE
			nState := 40; 
		END_IF
	END_IF	
	
	40:
	IF fbSqlResult.Read(0, 10000, ADR(DataRead), SIZEOF(DataRead), FALSE, TRUE) THEN
		IF fbSqlResult.bError THEN
			nState := 253; 
		ELSE
			nState := 50; 
		END_IF
	END_IF
	
	50:
	
	fbSqlResult.Release();
	
	IF fbSqlResult.bError THEN
		nState := 254 ;
	ELSE
		nState := 60;	
	END_IF

	
	60: 	
	fbSqlResult.Release();	
	
	IF fbSqlDatabase.Disconnect() THEN
		IF fbSqlDatabase.bError THEN
			nState := 255;
		ELSE
			nState := 0;
   		END_IF
	END_IF

250: ;
251: ;
252: ;
253: ;
254: ;
255: ;
	
END_CASE

END_FUNCTION_BLOCK

// ---- FCs/FC_ConcatStr.TcPOU
FUNCTION FC_ConcatStr : STRING(1500)
VAR_INPUT
	str1 : STRING(1500);
	str2 : STRING(1500);
END_VAR
VAR
	size1 : INT;
	size2 : INT;
	i : INT;
	j : INT;
END_VAR

size1 := 0;
size2 := 0;
FOR i := 0 TO 1500 BY 1 DO
	IF str1[i] = 0 THEN
		EXIT;
	ELSE
		size1 := size1 + 1;
	END_IF
END_FOR

FOR i := 0 TO 1500 BY 1 DO
	IF str2[i] = 0 THEN
		EXIT;
	ELSE
		size2 := size2 + 1;
	END_IF
END_FOR

FOR i := 0 TO 1500 BY 1 DO
	IF i < size1 THEN
		FC_ConcatStr[i] := str1[i];
	ELSIF i < size1 + size2 THEN
		FC_ConcatStr[i] := str2[i - size1];
	ELSE
		FC_ConcatStr[i] := 0;
	END_IF;
END_FOR

END_FUNCTION

// ---- FBs/Database/General/FB_SQL_ReadWithData.TcPOU
FUNCTION_BLOCK FB_SQL_ReadWithData
VAR_INPUT
	bExecute : BOOL ;	
	hDBID : UDINT 	:= 1;
	sSqlCommand: STRING(1000);	
END_VAR
VAR_OUTPUT
	aData : ARRAY[0..10000] OF ST_DatabasePower ;
END_VAR
VAR
	fbSqlDatabase : FB_SQLDatabaseEvt(sNetID := '', tTimeout := T#180S);
	fbSqlCommand : FB_SQLCommandEvt(sNetID := '', tTimeout := T#180S) ;
    fbSqlResult : FB_SQLResultEvt(sNetID:='', tTimeout    := T#180S); 
	fbPulse : R_TRIG ;	
	sDateStartAux : STRING ;	
	sDateEndtAux : STRING ;	
	nState: INT;
		
END_VAR

(* Pulso de uma varredura *)
fbPulse(CLK:= bExecute, Q=> );

IF fbPulse.Q THEN
	nState := 10 ;
END_IF
	
CASE nState OF

0:
//Iddle
;

10:

IF fbSqlDatabase.Connect(hDBID) THEN
	IF fbSqlDatabase.bError THEN
		nState := 250; 
	ELSE
		nState := 20; 
	END_IF
END_IF

20:	
IF fbSqlDatabase.CreateCmd(ADR(fbSqlCommand)) THEN
	IF fbSqlDatabase.bError THEN
		nState := 251; 
	ELSE
		nState := 30; 
	END_IF
END_IF	


30:

IF fbSqlCommand.ExecuteDataReturn(pSQLCmd:= ADR(sSqlCommand), cbSQLCmd:= SIZEOF(sSqlCommand), pSQLDBResult:= ADR(aData) ) THEN


	IF fbSQLCommand.bError THEN
		nState := 252; 
	ELSE
		nState := 40; 
	END_IF
END_IF	


40:

IF fbSqlResult.Read(nStartIndex:= 1, nRecordCount:= 1000, pData:= ADR(aData), cbData:= SIZEOF(aData), bWithVerifying:= FALSE , bDataRelease:= TRUE) THEN
	IF fbSqlResult.bError THEN
        nState := 253; 
    ELSE
        nState := 50; 
    END_IF
END_IF


50:

 IF fbSqlResult.Release() THEN
	IF fbSqlResult.bError THEN
		nState := 254 ;
	ELSE
		nState := 60;	
	END_IF
END_IF

60: 	

IF fbSqlDatabase.Disconnect() THEN
	IF fbSqlDatabase.bError THEN
		nState := 255;
	ELSE
		nState := 0;
	END_IF
END_IF

250: ;
251: ;
252: ;
253: ;
254: ;
255: ;
	
END_CASE

END_FUNCTION_BLOCK

// ---- FBs/Database/General/FB_SQL_TO_CSV.TcPOU
FUNCTION_BLOCK FB_SQL_TO_CSV
VAR_INPUT
	bExecute : BOOL ;
END_VAR
VAR_OUTPUT
END_VAR
VAR
	hDBID : UDINT 	:= 1;
	fbSqlDatabase : FB_SQLDatabaseEvt(sNetID := '', tTimeout := T#180S);
	fbSqlCommand : FB_SQLCommandEvt(sNetID := '', tTimeout := T#180S) ;
    fbSqlResult : FB_SQLResultEvt(sNetID:='', tTimeout    := T#180S); 
	fbPulse : R_TRIG ;	
	sDateStartAux : STRING ;	
	sDateEndtAux : STRING ;	
	nState: INT;
	sSqlCommand: STRING(INT#450);
END_VAR



sSqlCommand := 'DECLARE @SQLQuery AS NVARCHAR(200) 
				DECLARE @FilePath AS NVARCHAR(200)  
				SET @SQLQuery = $'SELECT * FROM [DB_PowerMeasure].[dbo].[TB_PowerMeter]$'
				SET @FilePath = $'C:\temp\arquivo.csv$' 
				SET @SQLQuery = $'bcp "$' + @SQLQuery + $'" queryout "$' + @FilePath + $'" -c -t, -T -S DOUGLASC-NB01\SQLEXPRESS$'  
				EXEC xp_cmdshell @SQLQuery  ';

fbPulse(CLK:= bExecute, Q=> );


IF fbPulse.Q THEN
	nState := 10 ;
END_IF
	


CASE nState OF

0:

;

10:

IF fbSqlDatabase.Connect(hDBID) THEN
	IF fbSqlDatabase.bError THEN
		nState := 250; 
	ELSE
		nState := 20; 
	END_IF
END_IF

20:	
IF fbSqlDatabase.CreateCmd(ADR(fbSqlCommand)) THEN
	IF fbSqlDatabase.bError THEN
		nState := 251; 
	ELSE
		nState := 30; 
	END_IF
END_IF	


30:
IF fbSqlCommand.Execute(pSQLCmd:= ADR(sSqlCommand), cbSQLCmd:= SIZEOF(sSqlCommand)) THEN

	IF fbSQLCommand.bError THEN
		nState := 252; 
	ELSE
		nState := 40; 
	END_IF
END_IF	


40:

fbSqlResult.Release();

IF fbSqlResult.bError THEN
	nState := 254 ;
ELSE
	nState := 50;	
END_IF


50: 	
fbSqlResult.Release();	

IF fbSqlDatabase.Disconnect() THEN
	IF fbSqlDatabase.bError THEN
		nState := 255;
	ELSE
		nState := 0;
	END_IF
END_IF

250: ;
251: ;
252: ;
253: ;
254: ;
255: ;
	
END_CASE

END_FUNCTION_BLOCK

// ---- FBs/Process/FB_Pump.TcPOU
FUNCTION_BLOCK FB_Pump
VAR_INPUT
	command : BOOL ;
	feedback : BOOL ;
	auto_man : BOOL ;
	time_feedback : INT ;
END_VAR
VAR_OUTPUT
	valve: BOOL;	
END_VAR
VAR
	fbTimer: TON;
	fail : BOOL ;
END_VAR

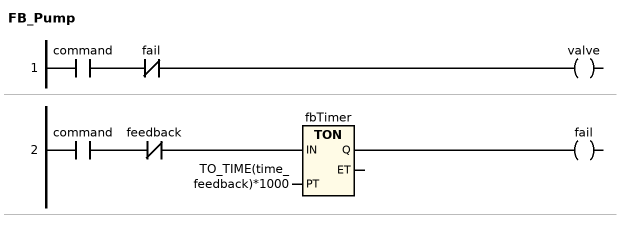
// NETWORK 1
valve := command AND NOT fail;

// NETWORK 2
fbTimer(IN := command AND NOT feedback, PT := TO_TIME(time_feedback)*1000); // TON
fail := fbTimer.Q;

END_FUNCTION_BLOCK

// ---- FBs/Process/FB_Valve.TcPOU
FUNCTION_BLOCK FB_Valve
VAR_INPUT
	command : BOOL ;
	feedback : BOOL ;
	auto_man : BOOL ;
	time_feedback : INT ;
END_VAR
VAR_OUTPUT
	valve: BOOL;	
END_VAR
VAR
	fbTimer: TON;
	fail : BOOL ;
END_VAR

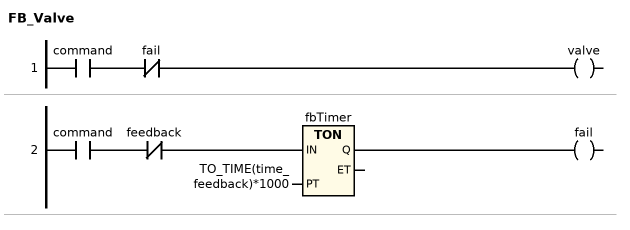
// NETWORK 1
valve := command AND NOT fail;

// NETWORK 2
fbTimer(IN := command AND NOT feedback, PT := TO_TIME(time_feedback)*1000); // TON
fail := fbTimer.Q;

END_FUNCTION_BLOCK

// ---- POUs/Eletric/PRG_Eletric.TcPOU
PROGRAM PRG_Eletric
VAR
END_VAR

END_PROGRAM

// ---- POUs/Process/PRG_Process.TcPOU
PROGRAM PRG_Process
VAR
	iTank : INT ;
END_VAR




iTank := iTank + 1 ;

END_PROGRAM
